// TIA Portal V18 export
FUNCTION_BLOCK "execute_semiauto"   // FB46, FBD
{ S7_Optimized_Access := 'TRUE' }
VERSION : 0.1
// stored: AutoNumber true, IsIECCheckEnabled false, IsRetainMemResEnabled false, MemoryReserve 100, SetENOAutomatically false, UDAEnableTagReadback false
   VAR_INPUT
      ALLOWED : Bool;
      xButton : Bool;
      arrived : Bool;
   END_VAR
   VAR_OUTPUT
      y_exec : Bool;
   END_VAR
   VAR
      mem : Bool;
      R_TRIG_Instance { S7_SetPoint := 'True'} : R_TRIG;
      loc : Bool;
   END_VAR
BEGIN

REGION Network 2 (SCL)
   #R_TRIG_Instance(CLK := #xButton);
   IF #ALLOWED THEN
       #y_exec := true;
   (*    IF #R_TRIG_Instance.Q THEN
           IF NOT #arrived THEN
               #y_exec := true;
           ELSE
               #y_exec := false;
           END_IF;
       END_IF; *)
   ELSE
       #y_exec := false;
   END_IF;
END_REGION
END_FUNCTION_BLOCK
